ABB RAPID module: GM2698_A.mod

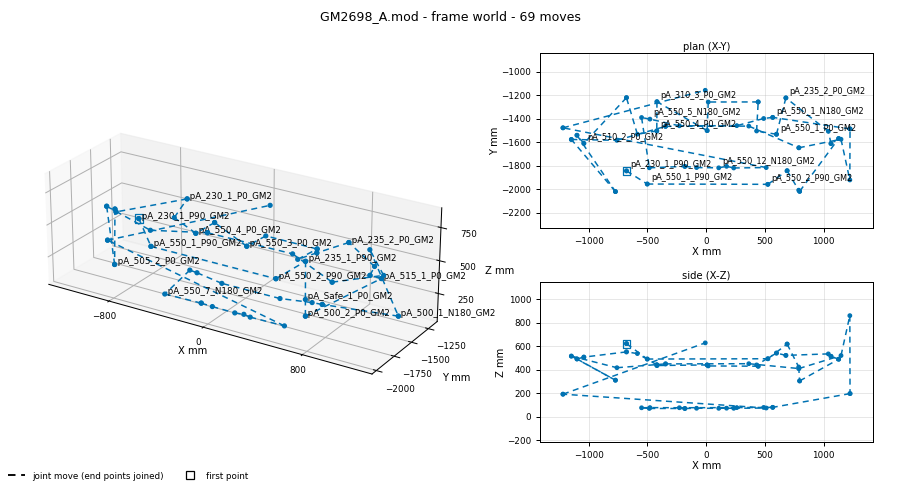
[picture p0: tool path of GM2698_A.mod in frame world, 69 of 75 moves have a stored position in this frame; points joined in program order, loops and branches not executed]
MODULE GM2698_A
!Tool number 7
	TASK PERS wobjdata wobj_A_GM2:=[FALSE,TRUE,"STN2",[[13.9887,-1106.54,385.608],[0.000303697,0.000861464,0.00233511,0.999997]],[[5.18442,-1.41215,-6.83269],[0.999989,-0.00459694,0.000966028,0.00104401]]];

	CONST robtarget pGM2698Tool_A_X1_GM2:=[[548.29,-1104.36,378.90],[0.999992,7.82758E-05,-0.000104085,0.00393794],[-1,0,-1,1],[9E+09,9E+09,9E+09,9E+09,0.0286518,9E+09]];
	CONST robtarget pGM2698Tool_A_X2_GM2:=[[-529.79,-1105.95,378.66],[1,1.60933E-06,-2.29478E-05,2.63453E-05],[-2,-1,0,1],[9E+09,9E+09,9E+09,9E+09,0.0293692,9E+09]];
	CONST robtarget pGM2698Tool_A_Y1_GM2:=[[10.44,-2216.22,373.75],[1,-3.56138E-05,-7.66218E-05,9.50694E-06],[-1,0,-1,1],[9E+09,9E+09,9E+09,9E+09,0.414757,9E+09]];

	!!TRUNNION AT P90
	CONST robtarget pA_230_1_P90_GM2:=[[687.93,736.01,247.05],[8.58268E-05,2.46025E-05,0.000125716,-1],[-2,-1,0,1],[9E+09,9E+09,9E+09,9E+09,89.9785,9E+09]];
	CONST robtarget pA_230_2_P90_GM2:=[[708.26,975.31,-115.95],[0.037863,-0.00102003,-0.000432508,-0.999282],[-2,-1,0,1],[9E+09,9E+09,9E+09,9E+09,44.9633,9E+09]];
	CONST robtarget pA_230_3_P90_GM2:=[[708.26,975.31,-115.95],[0.037863,-0.00102003,-0.000432508,-0.999282],[-2,-1,0,1],[9E+09,9E+09,9E+09,9E+09,44.9633,9E+09]];
	!
	CONST robtarget pA_235_1_P90_GM2:=[[-678.61,736.57,242.76],[0.00931104,0.000190613,-8.92784E-05,0.999957],[-1,0,-1,1],[9E+09,9E+09,9E+09,9E+09,89.9715,9E+09]];
	CONST robtarget pA_235_2_P90_GM2:=[[708.26,975.31,-115.95],[0.037863,-0.00102003,-0.000432508,-0.999282],[-2,-1,0,1],[9E+09,9E+09,9E+09,9E+09,44.9633,9E+09]];
	CONST robtarget pA_235_3_P90_GM2:=[[708.26,975.31,-115.95],[0.037863,-0.00102003,-0.000432508,-0.999282],[-2,-1,0,1],[9E+09,9E+09,9E+09,9E+09,44.9633,9E+09]];
	!
	CONST robtarget pA_310_1_P90_GM2:=[[353.10,729.89,294.43],[0.000108228,5.31787E-05,0.0438261,0.999039],[-2,-1,0,1],[9E+09,9E+09,9E+09,9E+09,89.9716,9E+09]];
	CONST robtarget pA_310_2_P90_GM2:=[[120.58,746.64,293.48],[0.000119282,2.78364E-05,-0.0697897,0.997561],[-2,-1,0,1],[9E+09,9E+09,9E+09,9E+09,89.9659,9E+09]];
	CONST robtarget pA_310_3_P90_GM2:=[[-126.06,745.90,293.24],[8.89304E-05,2.54854E-06,-0.0697908,0.997561],[-1,0,-1,1],[9E+09,9E+09,9E+09,9E+09,89.9658,9E+09]];
	CONST robtarget pA_310_4_P90_GM2:=[[-352.83,729.33,296.03],[0.000103667,2.41673E-05,0.0452051,0.998978],[-1,0,-1,1],[9E+09,9E+09,9E+09,9E+09,89.9674,9E+09]];
	CONST robtarget pA_310_5_P90_GM2:=[[708.26,975.31,-115.95],[0.037863,-0.00102003,-0.000432508,-0.999282],[-2,-1,0,1],[9E+09,9E+09,9E+09,9E+09,44.9633,9E+09]];
	!
	CONST robtarget pA_550_1_P90_GM2:=[[511.36,848.54,116.26],[0.000118797,-6.09284E-05,3.87415E-05,-1],[-2,-1,0,1],[9E+09,9E+09,9E+09,9E+09,89.9792,9E+09]];
	CONST robtarget pA_550_2_P90_GM2:=[[-514.41,852.57,118.58],[0.000364177,0.00017202,0.00027161,-1],[-1,0,-1,1],[9E+09,9E+09,9E+09,9E+09,89.9758,9E+09]];
	CONST robtarget pA_550_3_P90_GM2:=[[335.13,751.81,293.47],[0.000114739,1.47188E-05,-0.069799,0.997561],[-2,-1,0,1],[9E+09,9E+09,9E+09,9E+09,89.9654,9E+09]];
	CONST robtarget pA_550_4_P90_GM2:=[[335.13,751.81,293.47],[0.000114739,1.47188E-05,-0.069799,0.997561],[-2,-1,0,1],[9E+09,9E+09,9E+09,9E+09,89.9654,9E+09]];
	CONST robtarget pA_550_5_P90_GM2:=[[335.13,751.81,293.47],[0.000114739,1.47188E-05,-0.069799,0.997561],[-2,-1,0,1],[9E+09,9E+09,9E+09,9E+09,89.9654,9E+09]];
	CONST robtarget pA_550_6_P90_GM2:=[[335.13,751.81,293.47],[0.000114739,1.47188E-05,-0.069799,0.997561],[-2,-1,0,1],[9E+09,9E+09,9E+09,9E+09,89.9654,9E+09]];
	CONST robtarget pA_550_7_P90_GM2:=[[335.13,751.81,293.47],[0.000114739,1.47188E-05,-0.069799,0.997561],[-2,-1,0,1],[9E+09,9E+09,9E+09,9E+09,89.9654,9E+09]];
	CONST robtarget pA_550_8_P90_GM2:=[[335.13,751.81,293.47],[0.000114739,1.47188E-05,-0.069799,0.997561],[-2,-1,0,1],[9E+09,9E+09,9E+09,9E+09,89.9654,9E+09]];
	CONST robtarget pA_550_9_P90_GM2:=[[335.13,751.81,293.47],[0.000114739,1.47188E-05,-0.069799,0.997561],[-2,-1,0,1],[9E+09,9E+09,9E+09,9E+09,89.9654,9E+09]];
	CONST robtarget pA_550_10_P90_GM2:=[[335.13,751.81,293.47],[0.000114739,1.47188E-05,-0.069799,0.997561],[-2,-1,0,1],[9E+09,9E+09,9E+09,9E+09,89.9654,9E+09]];

	!!TRUNNION AT P0
	CONST robtarget pA_230_1_P0_GM2:=[[687.38,113.52,173.86],[0.00744481,0.444927,0.0139379,-0.895428],[-2,-1,-1,1],[9E+09,9E+09,9E+09,9E+09,-0.0044309,9E+09]];
	CONST robtarget pA_230_2_P0_GM2:=[[714.73,248.80,217.03],[0.0301629,0.281201,0.193711,0.939411],[-2,-2,1,1],[9E+09,9E+09,9E+09,9E+09,14.3078,9E+09]];
	CONST robtarget pA_230_3_P0_GM2:=[[708.26,975.31,-115.95],[0.037863,-0.00102003,-0.000432508,-0.999282],[-2,-1,0,1],[9E+09,9E+09,9E+09,9E+09,44.9633,9E+09]];
	!
	CONST robtarget pA_235_1_P0_GM2:=[[-730.47,258.27,215.19],[0.0469032,0.293033,-0.14088,-0.944503],[-1,1,-2,1],[9E+09,9E+09,9E+09,9E+09,15.4894,9E+09]];
	CONST robtarget pA_235_2_P0_GM2:=[[-668.80,117.45,143.98],[0.00289527,-0.436527,-0.00432652,-0.899677],[-1,0,0,1],[9E+09,9E+09,9E+09,9E+09,-0.011942,9E+09]];
	CONST robtarget pA_235_3_P0_GM2:=[[708.26,975.31,-115.95],[0.037863,-0.00102003,-0.000432508,-0.999282],[-2,-1,0,1],[9E+09,9E+09,9E+09,9E+09,44.9633,9E+09]];
	!
	CONST robtarget pA_310_1_P0_GM2:=[[-433.18,151.92,51.95],[1.60386E-05,5.67962E-05,0.0413145,0.999146],[-1,0,-1,1],[9E+09,9E+09,9E+09,9E+09,-0.0118576,9E+09]];
	CONST robtarget pA_310_2_P0_GM2:=[[-8.33,151.75,54.29],[6.56249E-05,0.000101471,0.0457973,0.998951],[-1,0,-1,1],[9E+09,9E+09,9E+09,9E+09,-0.0110137,9E+09]];
	CONST robtarget pA_310_3_P0_GM2:=[[428.07,148.75,57.96],[2.66549E-05,-6.70695E-06,0.0471647,0.998887],[-2,-1,0,1],[9E+09,9E+09,9E+09,9E+09,-0.00898821,9E+09]];
	CONST robtarget pA_310_4_P0_GM2:=[[708.26,975.31,-115.95],[0.037863,-0.00102003,-0.000432508,-0.999282],[-2,-1,0,1],[9E+09,9E+09,9E+09,9E+09,44.9633,9E+09]];
	CONST robtarget pA_310_5_P0_GM2:=[[708.26,975.31,-115.95],[0.037863,-0.00102003,-0.000432508,-0.999282],[-2,-1,0,1],[9E+09,9E+09,9E+09,9E+09,44.9633,9E+09]];
	!
	CONST robtarget pA_500_1_P0_GM2:=[[-1201.57,789.37,-64.62],[0.00293341,-0.00121104,0.000140597,-0.999995],[-1,0,-1,1],[9E+09,9E+09,9E+09,9E+09,29.7666,9E+09]];
	CONST robtarget pA_500_2_P0_GM2:=[[-784.67,913.62,-69.87],[0.0310443,0.0713657,0.0170151,-0.996822],[-1,0,-1,1],[9E+09,9E+09,9E+09,9E+09,29.7701,9E+09]];
	CONST robtarget pA_500_3_P0_GM2:=[[708.26,975.31,-115.95],[0.037863,-0.00102003,-0.000432508,-0.999282],[-2,-1,0,1],[9E+09,9E+09,9E+09,9E+09,44.9633,9E+09]];
	CONST robtarget pA_500_4_P0_GM2:=[[708.26,975.31,-115.95],[0.037863,-0.00102003,-0.000432508,-0.999282],[-2,-1,0,1],[9E+09,9E+09,9E+09,9E+09,44.9633,9E+09]];
	CONST robtarget pA_500_5_P0_GM2:=[[708.26,975.31,-115.95],[0.037863,-0.00102003,-0.000432508,-0.999282],[-2,-1,0,1],[9E+09,9E+09,9E+09,9E+09,44.9633,9E+09]];
	!
	CONST robtarget pA_505_1_P0_GM2:=[[1202.97,791.70,-68.86],[0.00492061,0.00110187,-4.76185E-05,0.999987],[-2,-1,0,1],[9E+09,9E+09,9E+09,9E+09,29.4165,9E+09]];
	CONST robtarget pA_505_2_P0_GM2:=[[782.38,913.28,-63.33],[0.0152789,0.0774775,-0.00477043,0.996866],[-2,-1,0,1],[9E+09,9E+09,9E+09,9E+09,29.4215,9E+09]];
	CONST robtarget pA_505_3_P0_GM2:=[[708.26,975.31,-115.95],[0.037863,-0.00102003,-0.000432508,-0.999282],[-2,-1,0,1],[9E+09,9E+09,9E+09,9E+09,44.9633,9E+09]];
	CONST robtarget pA_505_4_P0_GM2:=[[708.26,975.31,-115.95],[0.037863,-0.00102003,-0.000432508,-0.999282],[-2,-1,0,1],[9E+09,9E+09,9E+09,9E+09,44.9633,9E+09]];
	CONST robtarget pA_505_5_P0_GM2:=[[708.26,975.31,-115.95],[0.037863,-0.00102003,-0.000432508,-0.999282],[-2,-1,0,1],[9E+09,9E+09,9E+09,9E+09,44.9633,9E+09]];
	!
	CONST robtarget pA_510_1_P0_GM2:=[[1108.89,432.68,115.17],[0.112654,0.176226,0.0162339,0.977748],[-2,-1,1,1],[9E+09,9E+09,9E+09,9E+09,-0.0107183,9E+09]];
	CONST robtarget pA_510_2_P0_GM2:=[[1050.40,501.98,131.19],[0.0176776,-0.325143,0.0102617,0.945444],[-2,-1,-1,1],[9E+09,9E+09,9E+09,9E+09,-0.0104229,9E+09]];
	CONST robtarget pA_510_3_P0_GM2:=[[1153.27,592.76,100.47],[0.0365802,0.172145,-0.0278504,0.983998],[-2,-1,1,1],[9E+09,9E+09,9E+09,9E+09,26.5127,9E+09]];
	CONST robtarget pA_510_4_P0_GM2:=[[1048.95,504.25,129.99],[0.0176891,-0.325131,0.010239,0.945448],[-2,-1,0,1],[9E+09,9E+09,9E+09,9E+09,-0.011562,9E+09]];
	!
	CONST robtarget pA_515_1_P0_GM2:=[[-1117.17,463.93,112.66],[0.108166,0.211616,-0.00270155,-0.971345],[-1,0,-2,1],[9E+09,9E+09,9E+09,9E+09,-0.012828,9E+09]];
	CONST robtarget pA_515_2_P0_GM2:=[[-1052.07,506.56,137.57],[0.000402809,-0.35302,0.000389817,-0.935616],[-1,0,0,1],[9E+09,9E+09,9E+09,9E+09,-0.0197907,9E+09]];
	CONST robtarget pA_515_3_P0_GM2:=[[-1152.24,635.08,93.24],[0.0988859,0.169779,0.00503263,-0.980495],[-1,0,-2,1],[9E+09,9E+09,9E+09,9E+09,36.5012,9E+09]];
	CONST robtarget pA_515_4_P0_GM2:=[[-1045.41,506.20,133.06],[0.000367603,-0.353062,0.000351063,-0.9356],[-1,0,0,1],[9E+09,9E+09,9E+09,9E+09,-0.0197905,9E+09]];
	!
	CONST robtarget pA_520_1_P0_GM2:=[[708.26,975.31,-115.95],[0.037863,-0.00102003,-0.000432508,-0.999282],[-2,-1,0,1],[9E+09,9E+09,9E+09,9E+09,44.9633,9E+09]];
	CONST robtarget pA_520_2_P0_GM2:=[[708.26,975.31,-115.95],[0.037863,-0.00102003,-0.000432508,-0.999282],[-2,-1,0,1],[9E+09,9E+09,9E+09,9E+09,44.9633,9E+09]];
	CONST robtarget pA_520_3_P0_GM2:=[[708.26,975.31,-115.95],[0.037863,-0.00102003,-0.000432508,-0.999282],[-2,-1,0,1],[9E+09,9E+09,9E+09,9E+09,44.9633,9E+09]];
	CONST robtarget pA_520_4_P0_GM2:=[[708.26,975.31,-115.95],[0.037863,-0.00102003,-0.000432508,-0.999282],[-2,-1,0,1],[9E+09,9E+09,9E+09,9E+09,44.9633,9E+09]];
	CONST robtarget pA_520_5_P0_GM2:=[[708.26,975.31,-115.95],[0.037863,-0.00102003,-0.000432508,-0.999282],[-2,-1,0,1],[9E+09,9E+09,9E+09,9E+09,44.9633,9E+09]];
	!
	CONST robtarget pA_550_1_P0_GM2:=[[-588.27,426.70,164.89],[0.0152053,0.548166,0.0110567,0.836158],[-2,0,0,1],[9E+09,9E+09,9E+09,9E+09,-0.0169634,9E+09]];
	CONST robtarget pA_550_2_P0_GM2:=[[-419.34,398.83,64.09],[1.55675E-05,-3.99913E-05,1.7675E-05,1],[-1,0,-1,1],[9E+09,9E+09,9E+09,9E+09,-0.0173011,9E+09]];
	CONST robtarget pA_550_3_P0_GM2:=[[1.46,395.01,63.93],[1.08108E-05,-9.40457E-06,-2.05058E-05,-1],[-1,0,-1,1],[9E+09,9E+09,9E+09,9E+09,-0.022618,9E+09]];
	CONST robtarget pA_550_4_P0_GM2:=[[429.81,397.20,65.70],[8.27019E-06,8.95741E-05,-5.33681E-05,1],[-2,-1,0,1],[9E+09,9E+09,9E+09,9E+09,-0.0133345,9E+09]];
	CONST robtarget pA_550_5_P0_GM2:=[[594.89,424.65,160.92],[0.028073,0.537019,-0.0220339,-0.842814],[-1,-1,-1,1],[9E+09,9E+09,9E+09,9E+09,-0.0155708,9E+09]];
	CONST robtarget pA_550_6_P0_GM2:=[[708.26,975.31,-115.95],[0.037863,-0.00102003,-0.000432508,-0.999282],[-2,-1,0,1],[9E+09,9E+09,9E+09,9E+09,44.9633,9E+09]];
	CONST robtarget pA_550_7_P0_GM2:=[[708.26,975.31,-115.95],[0.037863,-0.00102003,-0.000432508,-0.999282],[-2,-1,0,1],[9E+09,9E+09,9E+09,9E+09,44.9633,9E+09]];
	CONST robtarget pA_550_8_P0_GM2:=[[708.26,975.31,-115.95],[0.037863,-0.00102003,-0.000432508,-0.999282],[-2,-1,0,1],[9E+09,9E+09,9E+09,9E+09,44.9633,9E+09]];
	CONST robtarget pA_550_9_P0_GM2:=[[708.26,975.31,-115.95],[0.037863,-0.00102003,-0.000432508,-0.999282],[-2,-1,0,1],[9E+09,9E+09,9E+09,9E+09,44.9633,9E+09]];
	CONST robtarget pA_550_10_P0_GM2:=[[708.26,975.31,-115.95],[0.037863,-0.00102003,-0.000432508,-0.999282],[-2,-1,0,1],[9E+09,9E+09,9E+09,9E+09,44.9633,9E+09]];
	!
	!!TRUNNION AT N60
	CONST robtarget pA_500_1_N60_GM2:=[[-778.58,542.42,33.75],[0.00280107,0.0438531,0.00715282,-0.999009],[-1,0,-1,1],[9E+09,9E+09,9E+09,9E+09,-60.5132,9E+09]];
	CONST robtarget pA_500_2_N60_GM2:=[[-1217.46,473.19,8.92],[0.00374905,-0.104264,0.00695893,-0.994518],[-1,0,-1,1],[9E+09,9E+09,9E+09,9E+09,-60.5084,9E+09]];
	CONST robtarget pA_500_3_N60_GM2:=[[-1137.33,470.02,143.84],[0.00403999,-0.000135764,2.34192E-05,-0.999992],[-1,0,-1,1],[9E+09,9E+09,9E+09,9E+09,-60.5103,9E+09]];
	CONST robtarget pA_500_4_N60_GM2:=[[708.26,975.31,-115.95],[0.037863,-0.00102003,-0.000432508,-0.999282],[-2,-1,0,1],[9E+09,9E+09,9E+09,9E+09,44.9633,9E+09]];
	CONST robtarget pA_500_5_N60_GM2:=[[708.26,975.31,-115.95],[0.037863,-0.00102003,-0.000432508,-0.999282],[-2,-1,0,1],[9E+09,9E+09,9E+09,9E+09,44.9633,9E+09]];
	!
	CONST robtarget pA_505_1_N60_GM2:=[[1156.75,468.38,139.62],[0.00522979,-1.17706E-05,-7.50595E-05,-0.999987],[-2,-1,0,1],[9E+09,9E+09,9E+09,9E+09,-60.5089,9E+09]];
	CONST robtarget pA_505_2_N60_GM2:=[[1216.37,472.20,8.95],[0.00194678,0.139228,0.00768064,-0.990228],[-2,-1,0,1],[9E+09,9E+09,9E+09,9E+09,-60.506,9E+09]];
	CONST robtarget pA_505_3_N60_GM2:=[[769.08,476.65,40.85],[0.0019964,-0.0777815,-8.25469E-05,-0.996969],[-2,-1,0,1],[9E+09,9E+09,9E+09,9E+09,-60.5041,9E+09]];
	CONST robtarget pA_505_4_N60_GM2:=[[708.26,975.31,-115.95],[0.037863,-0.00102003,-0.000432508,-0.999282],[-2,-1,0,1],[9E+09,9E+09,9E+09,9E+09,44.9633,9E+09]];
	CONST robtarget pA_505_5_N60_GM2:=[[708.26,975.31,-115.95],[0.037863,-0.00102003,-0.000432508,-0.999282],[-2,-1,0,1],[9E+09,9E+09,9E+09,9E+09,44.9633,9E+09]];
	!
	CONST robtarget pA_520_1_N60_GM2:=[[355.07,358.37,72.76],[0.00521062,-0.000565034,0.105165,-0.994441],[-2,-1,0,1],[9E+09,9E+09,9E+09,9E+09,-60.5116,9E+09]];
	CONST robtarget pA_520_2_N60_GM2:=[[-123.90,988.17,-108.46],[0.000713776,4.54184E-05,8.43669E-05,-0.999999],[-1,0,-1,1],[9E+09,9E+09,9E+09,9E+09,60.0162,9E+09]];
	CONST robtarget pA_520_3_N60_GM2:=[[123.84,989.35,-108.45],[0.000730733,6.40844E-05,7.66397E-05,-0.999999],[-2,-1,0,1],[9E+09,9E+09,9E+09,9E+09,60.0163,9E+09]];
	CONST robtarget pA_520_4_N60_GM2:=[[-353.01,357.21,74.17],[0.00521171,-0.000602148,0.105152,-0.994442],[-1,0,-1,1],[9E+09,9E+09,9E+09,9E+09,-60.5086,9E+09]];
	!
	!!TRUNNION AT N180
	!
	CONST robtarget pA_310_1_N180_GM2:=[[-427.01,928.00,-352.17],[4.23949E-05,1.23545E-06,-0.117062,-0.993125],[-1,0,-1,1],[9E+09,9E+09,9E+09,9E+09,-171.335,9E+09]];
	CONST robtarget pA_310_2_N180_GM2:=[[-341.86,937.73,-374.62],[1.08478E-05,-1.53197E-05,6.13881E-05,-1],[-1,0,-1,1],[9E+09,9E+09,9E+09,9E+09,-171.333,9E+09]];
	CONST robtarget pA_310_3_N180_GM2:=[[-161.23,931.93,-349.80],[8.00821E-06,-4.37144E-05,-0.117485,-0.993075],[-1,0,-1,1],[9E+09,9E+09,9E+09,9E+09,-171.335,9E+09]];
	CONST robtarget pA_310_4_N180_GM2:=[[9.06,936.16,-374.68],[2.71618E-05,-1.9313E-05,-0.0604457,-0.998172],[-2,-1,0,1],[9E+09,9E+09,9E+09,9E+09,-171.334,9E+09]];
	CONST robtarget pA_310_5_N180_GM2:=[[157.83,928.08,-351.40],[4.23165E-05,-2.36973E-05,-0.117106,-0.99312],[-2,-1,0,1],[9E+09,9E+09,9E+09,9E+09,-171.335,9E+09]];
	CONST robtarget pA_310_6_N180_GM2:=[[431.92,925.50,-350.73],[4.91988E-05,-7.21662E-05,-0.117557,-0.993066],[-2,-1,0,1],[9E+09,9E+09,9E+09,9E+09,-171.335,9E+09]];
	CONST robtarget pA_310_7_N180_GM2:=[[492.88,939.60,-374.19],[4.56863E-05,-1.05492E-05,6.13342E-05,-1],[-2,-1,0,1],[9E+09,9E+09,9E+09,9E+09,-171.333,9E+09]];
	CONST robtarget pA_310_8_N180_GM2:=[[708.26,975.31,-115.95],[0.037863,-0.00102003,-0.000432508,-0.999282],[-2,-1,0,1],[9E+09,9E+09,9E+09,9E+09,44.9633,9E+09]];
	CONST robtarget pA_310_9_N180_GM2:=[[708.26,975.31,-115.95],[0.037863,-0.00102003,-0.000432508,-0.999282],[-2,-1,0,1],[9E+09,9E+09,9E+09,9E+09,44.9633,9E+09]];
	CONST robtarget pA_310_10_N180_GM2:=[[708.26,975.31,-115.95],[0.037863,-0.00102003,-0.000432508,-0.999282],[-2,-1,0,1],[9E+09,9E+09,9E+09,9E+09,44.9633,9E+09]];
	CONST robtarget pA_310_11_N180_GM2:=[[708.26,975.31,-115.95],[0.037863,-0.00102003,-0.000432508,-0.999282],[-2,-1,0,1],[9E+09,9E+09,9E+09,9E+09,44.9633,9E+09]];
	CONST robtarget pA_310_12_N180_GM2:=[[708.26,975.31,-115.95],[0.037863,-0.00102003,-0.000432508,-0.999282],[-2,-1,0,1],[9E+09,9E+09,9E+09,9E+09,44.9633,9E+09]];
	CONST robtarget pA_310_13_N180_GM2:=[[708.26,975.31,-115.95],[0.037863,-0.00102003,-0.000432508,-0.999282],[-2,-1,0,1],[9E+09,9E+09,9E+09,9E+09,44.9633,9E+09]];
	CONST robtarget pA_310_14_N180_GM2:=[[708.26,975.31,-115.95],[0.037863,-0.00102003,-0.000432508,-0.999282],[-2,-1,0,1],[9E+09,9E+09,9E+09,9E+09,44.9633,9E+09]];
	CONST robtarget pA_310_15_N180_GM2:=[[708.26,975.31,-115.95],[0.037863,-0.00102003,-0.000432508,-0.999282],[-2,-1,0,1],[9E+09,9E+09,9E+09,9E+09,44.9633,9E+09]];

	!
	CONST robtarget pA_500_1_N180_GM2:=[[-1214.15,383.59,-180.12],[0.706069,-6.54173E-05,-1.71735E-05,-0.708144],[-1,-1,0,1],[9E+09,9E+09,9E+09,9E+09,-149.959,9E+09]];
	CONST robtarget pA_500_2_N180_GM2:=[[-1204.66,381.86,-186.15],[0.32853,-6.5977E-06,4.28364E-05,-0.944493],[-1,0,-1,1],[9E+09,9E+09,9E+09,9E+09,-149.952,9E+09]];
	CONST robtarget pA_500_3_N180_GM2:=[[-1137.07,519.96,141.43],[0.00405737,-1.80252E-05,5.82048E-05,-0.999991],[-1,0,-1,1],[9E+09,9E+09,9E+09,9E+09,-60.5062,9E+09]];
	CONST robtarget pA_500_4_N180_GM2:=[[708.26,975.31,-115.95],[0.037863,-0.00102003,-0.000432508,-0.999282],[-2,-1,0,1],[9E+09,9E+09,9E+09,9E+09,44.9633,9E+09]];
	CONST robtarget pA_500_5_N180_GM2:=[[708.26,975.31,-115.95],[0.037863,-0.00102003,-0.000432508,-0.999282],[-2,-1,0,1],[9E+09,9E+09,9E+09,9E+09,44.9633,9E+09]];
	!
	CONST robtarget pA_505_1_N180_GM2:=[[1227.95,370.76,-184.70],[0.703813,2.0347E-05,-0.000363019,0.710385],[-2,0,-1,1],[9E+09,9E+09,9E+09,9E+09,-149.954,9E+09]];
	CONST robtarget pA_505_2_N180_GM2:=[[1191.41,389.44,-184.88],[0.320474,-4.84084E-05,-0.000382623,0.947257],[-2,-1,0,1],[9E+09,9E+09,9E+09,9E+09,-149.948,9E+09]];
	CONST robtarget pA_505_3_N180_GM2:=[[775.04,447.88,42.59],[0.00201212,-0.0777562,-8.91676E-05,-0.99697],[-2,-1,0,1],[9E+09,9E+09,9E+09,9E+09,-60.5045,9E+09]];
	CONST robtarget pA_505_4_N180_GM2:=[[708.26,975.31,-115.95],[0.037863,-0.00102003,-0.000432508,-0.999282],[-2,-1,0,1],[9E+09,9E+09,9E+09,9E+09,44.9633,9E+09]];
	CONST robtarget pA_505_5_N180_GM2:=[[708.26,975.31,-115.95],[0.037863,-0.00102003,-0.000432508,-0.999282],[-2,-1,0,1],[9E+09,9E+09,9E+09,9E+09,44.9633,9E+09]];
	!
	CONST robtarget pA_550_1_N180_GM2:=[[-556.66,284.95,-297.43],[0.0146441,-0.000738703,-0.0640003,-0.997842],[-1,0,-1,1],[9E+09,9E+09,9E+09,9E+09,-179.982,9E+09]];
	CONST robtarget pA_550_2_N180_GM2:=[[-479.54,294.52,-298.21],[0.0147177,0.000968414,-0.0648092,-0.997788],[-1,0,-1,1],[9E+09,9E+09,9E+09,9E+09,-179.974,9E+09]];
	CONST robtarget pA_550_3_N180_GM2:=[[-250.78,354.86,-299.12],[0.00839662,0.00062424,-0.0673719,-0.997693],[-1,0,-1,1],[9E+09,9E+09,9E+09,9E+09,-179.978,9E+09]];
	CONST robtarget pA_550_4_N180_GM2:=[[237.67,355.52,-300.25],[0.006963,0.000448698,-0.0699319,-0.997528],[-2,-1,0,1],[9E+09,9E+09,9E+09,9E+09,-179.971,9E+09]];
	CONST robtarget pA_550_5_N180_GM2:=[[488.03,298.32,-299.34],[0.0147834,0.00108507,-0.0688852,-0.997515],[-2,-1,0,1],[9E+09,9E+09,9E+09,9E+09,-179.978,9E+09]];
	CONST robtarget pA_550_6_N180_GM2:=[[559.15,284.61,-300.90],[0.0147563,0.000914124,-0.0621348,-0.997959],[-2,-1,0,1],[9E+09,9E+09,9E+09,9E+09,-179.972,9E+09]];
	CONST robtarget pA_550_7_N180_GM2:=[[493.82,712.51,-304.58],[0.00369609,1.44225E-05,-0.000177454,0.999993],[-2,-1,0,1],[9E+09,9E+09,9E+09,9E+09,-179.978,9E+09]];
	CONST robtarget pA_550_8_N180_GM2:=[[191.37,701.01,-305.16],[0.000471327,-4.0688E-05,2.47394E-05,-1],[-2,-1,0,1],[9E+09,9E+09,9E+09,9E+09,-179.98,9E+09]];
	CONST robtarget pA_550_9_N180_GM2:=[[162.52,714.71,-304.99],[0.00044817,-2.64542E-05,3.82305E-05,-1],[-2,-1,0,1],[9E+09,9E+09,9E+09,9E+09,-179.977,9E+09]];
	CONST robtarget pA_550_10_N180_GM2:=[[92.00,710.92,-303.09],[0.000492036,-8.80391E-06,3.65271E-05,-1],[-2,-1,0,1],[9E+09,9E+09,9E+09,9E+09,-179.979,9E+09]];
	CONST robtarget pA_550_11_N180_GM2:=[[-2.18,734.80,-301.09],[0.000503616,-3.449E-05,2.8216E-05,-0.999999],[-2,0,-1,1],[9E+09,9E+09,9E+09,9E+09,-179.976,9E+09]];
	CONST robtarget pA_550_12_N180_GM2:=[[-96.61,713.50,-303.62],[0.000531659,-1.04945E-05,2.9268E-05,-1],[-1,0,-1,1],[9E+09,9E+09,9E+09,9E+09,-179.979,9E+09]];
	CONST robtarget pA_550_13_N180_GM2:=[[-163.24,700.92,-302.64],[0.000557157,-1.5553E-06,6.84997E-06,-1],[-1,0,-1,1],[9E+09,9E+09,9E+09,9E+09,-179.984,9E+09]];
	CONST robtarget pA_550_14_N180_GM2:=[[-224.30,714.89,-303.47],[0.000565679,-1.66874E-05,-1.44057E-05,-1],[-1,0,-1,1],[9E+09,9E+09,9E+09,9E+09,-179.982,9E+09]];
	CONST robtarget pA_550_15_N180_GM2:=[[-500.65,711.97,-301.26],[0.00055817,-3.54601E-05,1.56352E-05,-1],[-1,0,-1,1],[9E+09,9E+09,9E+09,9E+09,-179.988,9E+09]];
	CONST robtarget pA_550_16_N180_GM2:=[[335.13,751.81,293.47],[0.000114739,1.47188E-05,-0.069799,0.997561],[-2,-1,0,1],[9E+09,9E+09,9E+09,9E+09,89.9654,9E+09]];
	CONST robtarget pA_550_17_N180_GM2:=[[335.13,751.81,293.47],[0.000114739,1.47188E-05,-0.069799,0.997561],[-2,-1,0,1],[9E+09,9E+09,9E+09,9E+09,89.9654,9E+09]];
	CONST robtarget pA_550_18_N180_GM2:=[[335.13,751.81,293.47],[0.000114739,1.47188E-05,-0.069799,0.997561],[-2,-1,0,1],[9E+09,9E+09,9E+09,9E+09,89.9654,9E+09]];
	CONST robtarget pA_550_19_N180_GM2:=[[351.91,756.93,-300.99],[0.0147766,-2.34032E-05,6.93973E-05,-0.99989],[-2,-1,0,1],[9E+09,9E+09,9E+09,9E+09,-179.977,9E+09]];
	CONST robtarget pA_550_20_N180_GM2:=[[122.27,635.67,-305.15],[0.000474668,-1.23285E-05,1.97455E-05,-1],[-2,-1,0,1],[9E+09,9E+09,9E+09,9E+09,-179.978,9E+09]];
	CONST robtarget pA_550_21_N180_GM2:=[[-128.60,758.45,-301.12],[0.000539466,-5.17921E-06,1.67757E-05,-0.999999],[-1,0,-1,1],[9E+09,9E+09,9E+09,9E+09,-179.978,9E+09]];
	CONST robtarget pA_550_22_N180_GM2:=[[-356.72,760.25,-301.19],[0.000574946,-3.24014E-06,3.82912E-06,-0.999999],[-1,0,-1,1],[9E+09,9E+09,9E+09,9E+09,-179.98,9E+09]];


    TASK PERS loaddata LoadGM2698A:=[900,[-186.8,43.5,0],[1,0,0,0],0,0,111.6];


	CONST robtarget pA_Safe_1_P0_GM2:=[[-776.79,903.09,48.71],[0.0270915,0.0665119,0.0157283,-0.997294],[-1,0,-1,1],[9E+09,9E+09,9E+09,9E+09,31.3258,9E+09]];
	CONST robtarget pA_Safe_2_P0_GM2:=[[-1173.26,505.55,308.17],[0.299253,-0.00605452,0.0185665,-0.953974],[-1,0,-1,1],[9E+09,9E+09,9E+09,9E+09,-0.0127436,9E+09]];
	CONST robtarget pA_Safe_3_P0_GM2:=[[1206.65,483.09,309.68],[0.320571,-0.00610917,-0.0189757,0.947014],[-2,0,-1,1],[9E+09,9E+09,9E+09,9E+09,-0.012828,9E+09]];
	CONST robtarget pA_Safe_4_P0_GM2:=[[-867.31,489.74,258.29],[0.0101084,2.8178E-05,-5.44035E-05,0.999949],[-1,0,-1,1],[9E+09,9E+09,9E+09,9E+09,-0.012828,9E+09]];
	CONST robtarget pA_Safe_5_P0_GM2:=[[-867.31,489.74,258.29],[0.0101084,2.8178E-05,-5.44035E-05,0.999949],[-1,0,-1,1],[9E+09,9E+09,9E+09,9E+09,-0.012828,9E+09]];
	CONST robtarget pA_Safe_6_P0_GM2:=[[-867.31,489.74,258.29],[0.0101084,2.8178E-05,-5.44035E-05,0.999949],[-1,0,-1,1],[9E+09,9E+09,9E+09,9E+09,-0.012828,9E+09]];
	CONST robtarget pA_Safe_7_P0_GM2:=[[-867.31,489.74,258.29],[0.0101084,2.8178E-05,-5.44035E-05,0.999949],[-1,0,-1,1],[9E+09,9E+09,9E+09,9E+09,-0.012828,9E+09]];

	CONST robtarget pA_Safe_1_N180_GM2:=[[-1211.92,814.58,484.94],[0.113943,-0.0335182,0.225338,-0.967015],[-1,0,-1,1],[9E+09,9E+09,9E+09,9E+09,-62.6189,9E+09]];
	CONST robtarget pA_Safe_2_N180_GM2:=[[16.89,51.24,250.08],[0.00136107,-3.49227E-05,0.000388549,-0.999999],[-2,-1,0,1],[9E+09,9E+09,9E+09,9E+09,-149.948,9E+09]];
	CONST robtarget pA_Safe_3_N180_GM2:=[[16.88,51.24,250.08],[0.00136295,-3.96608E-05,0.000388216,-0.999999],[-2,-1,0,1],[9E+09,9E+09,9E+09,9E+09,33.5415,9E+09]];

	CONST robtarget pA_445_safe01_N180_GM2:=[[-1030.14,449.69,-57.42],[0.139634,-0.000906499,-0.000277604,-0.990202],[-1,0,-1,1],[9E+09,9E+09,9E+09,9E+09,-179.929,9E+09]];
	CONST robtarget pA_Safe_N90_2_GM2:=[[758.90,24.14,-68.10],[0.000305872,0.00120705,0.173796,0.98478],[-2,-1,0,1],[9E+09,9E+09,9E+09,9E+09,-58.1628,9E+09]];
	CONST robtarget pA_Safe_N90_3_GM2:=[[-894.81,518.59,346.96],[0.00406077,-2.99968E-05,5.05023E-05,-0.999991],[-1,0,-1,1],[9E+09,9E+09,9E+09,9E+09,-60.5068,9E+09]];
	CONST robtarget pA_Safe_1_P0_GM12:=[[-543.62,820.17,65.05],[5.02587E-05,0.000307266,5.46968E-06,1],[-1,0,-1,1],[9E+09,9E+09,9E+09,9E+09,-0.0227023,9E+09]];
	CONST robtarget pA_550_3_P0_GM12:=[[545.82,817.89,57.34],[2.78437E-05,0.000245156,0.000100892,1],[-2,-1,0,1],[9E+09,9E+09,9E+09,9E+09,-0.0315638,9E+09]];
	CONST robtarget pA_500_1_N180_GM12:=[[-1129.50,619.60,-361.57],[0.0233784,0.216958,0.0182336,0.97573],[-1,0,-1,1],[9E+09,9E+09,9E+09,9E+09,-178.615,9E+09]];
	CONST robtarget pA_515_1_P0_GM12:=[[-1117.17,463.93,112.66],[0.108168,0.211621,-0.00269871,-0.971344],[-1,0,-2,1],[9E+09,9E+09,9E+09,9E+09,-0.0123203,9E+09]];
	CONST robtarget pA_550_3_P0_GM22:=[[116.06,395.94,63.70],[3.88215E-05,-1.77326E-05,1.06229E-05,-1],[-2,-1,0,1],[9E+09,9E+09,9E+09,9E+09,-0.0232087,9E+09]];
	CONST robtarget pA_Safe_1_P0_GM22:=[[-116.20,396.03,64.22],[3.20058E-05,-2.53767E-05,1.70392E-05,-1],[-1,0,-1,1],[9E+09,9E+09,9E+09,9E+09,-0.0232087,9E+09]];
	CONST robtarget pA_515_2_P0_GM12:=[[-1029.51,402.17,157.71],[0.000353747,-0.353072,0.000348763,-0.935597],[-1,0,0,1],[9E+09,9E+09,9E+09,9E+09,-0.0192,9E+09]];




	PROC rGM2698_A_Welding()
			SetGO TaskActive, 1;
			rSpeed_Override;
			ClkReset clock_A_Weld_cycle;
			ClkStart clock_A_Weld_cycle;
			PulseDO\PLength:=2.0, WeldStarted;
			!
			PulseDO\PLength:=2.0, OpenCellAInnerDoor;

			ActUnit STN2;
			!DeactUnit STN1;
			MechUnitLoad Stn2, 1, LoadGM2698A;
			WaitDI CellAInnerDoorOpened ,1;
			!

		IF RobotProduction = 1 THEN
			vProduction := [7500,7500,7500,180];
			vHome := [3500, 3500, 3500, 90];
	  	ELSE
			vProduction := [200,100,100,20];
			vHome := [100, 100, 100, 10];
	  	ENDIF
			!
			WaitDI TAClampsSafePFO,1;
			rMoveToCell_A;
			Set PFOAirJet;
			!
			MoveAbsJ pA_Load\NoEOffs, vProduction, z200, t3D_PFO\WObj:=wobj0;
			PulseDO WeldStarted;
			Set LaserRequest;
			IF TAClampsSafePFO = 0 Stop;
			!
			AccSet 100,100;

			!**************************************************
			!Positioner at +90 degree
			!**************************************************
			MoveJ pA_230_1_P90_GM2,vProduction,fine,t3D_PFO\WObj:=wobj_A_GM2;
			IF AS350_1PP = 1 THEN !!!TA230XPP = 1 Then
			!K2 SP
			SetGO PFOProgReq, 312;
			SetGO LaserProgReq, 140;
			MoveJ pA_230_1_P90_GM2,vProduction,fine,t3D_PFO\WObj:=wobj_A_GM2;
			rPFO_Welding;
			!
			ENDIF
			!
			MoveJ pA_550_1_P90_GM2,vProduction,fine,t3D_PFO\WObj:=wobj_A_GM2;
			IF AW550PP = 1 THEN  !!! TA550PP = 1 Then
			!
			!K2 WD
			SetGO PFOProgReq, 112;
			SetGO LaserProgReq, 140;
			MoveJ pA_550_1_P90_GM2,vProduction,fine,t3D_PFO\WObj:=wobj_A_GM2;
			rPFO_Welding;
			!
			ENDIF

			MoveJ pA_550_2_P90_GM2,vProduction,fine,t3D_PFO\WObj:=wobj_A_GM2;
			IF AW550PP = 1 THEN  !!! TA550PP = 1 Then
			!
			!M2 WD
			SetGO PFOProgReq, 118;
			SetGO LaserProgReq, 140;
			MoveJ pA_550_2_P90_GM2,vProduction,fine,t3D_PFO\WObj:=wobj_A_GM2;
			rPFO_Welding;
			!
			ENDIF


			MoveJ pA_235_1_P90_GM2,vProduction,fine,t3D_PFO\WObj:=wobj_A_GM2;
			IF AS350_2PP = 1 THEN !!!  TA235XPP = 1 Then
			!M2 SP
			SetGO PFOProgReq, 318;
			SetGO LaserProgReq, 140;
			MoveJ pA_235_1_P90_GM2,vProduction,fine,t3D_PFO\WObj:=wobj_A_GM2;
			rPFO_Welding;
			!
			ENDIF
			!**************************************************
			!Trunnion at +0 degree
			!*************************************************

			MoveJ pA_Safe_1_P0_GM2, vProduction, z200, t3D_PFO\WObj:=wobj_A_GM2;

			MoveJ pA_500_2_P0_GM2,vProduction,fine,t3D_PFO\WObj:=wobj_A_GM2;
			IF AW500PP = 1 THEN !!! TA500PP = 1 Then

			!H5 WD
			SetGO PFOProgReq, 99;
			SetGO LaserProgReq, 140;
			MoveJ pA_500_2_P0_GM2,vProduction,fine,t3D_PFO\WObj:=wobj_A_GM2;
			rPFO_Welding;

			ENDIF
			!
			MoveJ pA_515_1_P0_GM2,vProduction,fine,t3D_PFO\WObj:=wobj_A_GM2;
			IF AW510_2PP = 1 THEN !!!  TA515 = 1 Then
			!
			!G1 G2-1 G2-2 WD
			SetGO LaserProgReq, 147;
			MoveJ pA_515_1_P0_GM2,vProduction,fine,t3D_PFO\WObj:=wobj_A_GM2;
			rPFO_Welding;
			!WaitTime 1.0;

			ENDIF


		MoveJ pA_515_2_P0_GM2, vProduction, fine, t3D_PFO\WObj:=wobj_A_GM2;
			IF AW510_2PP = 1 THEN !!!  TA515 = 1 Then

			!G3 WD
			SetGO PFOProgReq, 92;
			SetGO LaserProgReq, 140;
			MoveJ pA_515_2_P0_GM2, vProduction, fine, t3D_PFO\WObj:=wobj_A_GM2;
			rPFO_Welding;

			MoveJ pA_515_2_P0_GM12, vPRODUCTION, z200, t3D_PFO\WObj:=wobj_A_GM2;
			!
			ENDIF

			MoveJ pA_235_2_P0_GM2,vProduction,fine,t3D_PFO\WObj:=wobj_A_GM2;
			IF AS350_2PP = 1 THEN !!!  TA235XPP = 1 Then

			!F6 F7 F8 F9 F10
			SetGO LaserProgReq, 149;
			MoveJ pA_235_2_P0_GM2,vProduction,fine,t3D_PFO\WObj:=wobj_A_GM2;
			rPFO_Welding;
			!
			ENDIF

			MoveJ pA_550_1_P0_GM2,vProduction,fine,t3D_PFO\WObj:=wobj_A_GM2;
			IF AW550PP = 1 THEN  !!! TA550PP = 1 Then
			!
			!M3 M4 WD
			SetGO LaserProgReq, 161;
			MoveJ pA_550_1_P0_GM2,vProduction,fine,t3D_PFO\WObj:=wobj_A_GM2;
			rPFO_Welding;
			!
			!M1
			SetGO PFOProgReq, 117;
			SetGO LaserProgReq, 140;
			MoveJ pA_550_2_P0_GM2,vProduction,fine,t3D_PFO\WObj:=wobj_A_GM2;
			rPFO_Welding;
			!
			ENDIF

			MoveJ pA_310_1_P0_GM2,vProduction,fine,t3D_PFO\WObj:=wobj_A_GM2;

			IF AS310PP = 1 THEN !!! TA310XPP = 1 Then
			!K1 SP
			SetGO PFOProgReq, 311;
			SetGO LaserProgReq, 140;
			MoveJ pA_310_1_P0_GM2,vProduction,fine,t3D_PFO\WObj:=wobj_A_GM2;
			rPFO_Welding;
			!
			!J1 J2 SP
			SetGO PFOProgReq, 302;
			SetGO LaserProgReq, 140;
			MoveJ pA_310_2_P0_GM2,vProduction,fine,t3D_PFO\WObj:=wobj_A_GM2;
			rPFO_Welding;

			ENDIF

			MoveJ pA_550_3_P0_GM2,vProduction,fine,t3D_PFO\WObj:=wobj_A_GM2;
			IF AW550PP = 1 THEN  !!! TA550PP = 1 Then

			!J1 J2 WD
			SetGO LaserProgReq, 163;
			MoveJ pA_550_3_P0_GM2,vProduction,fine,t3D_PFO\WObj:=wobj_A_GM2;
			rPFO_Welding;

			ENDIF

			MoveJ pA_310_3_P0_GM2,vProduction,fine,t3D_PFO\WObj:=wobj_A_GM2;
			IF AS310PP = 1 THEN !!! TA310XPP = 1 Then
			!
			SetGO PFOProgReq, 317;
			SetGO LaserProgReq, 140;
			MoveJ pA_310_3_P0_GM2,vProduction,fine,t3D_PFO\WObj:=wobj_A_GM2;
			rPFO_Welding;
			!
			ENDIF

			MoveJ pA_550_4_P0_GM2,vProduction,fine,t3D_PFO\WObj:=wobj_A_GM2;
			IF AW550PP = 1 THEN  !!! TA550PP = 1 Then
			!
			!K1 WD
			SetGO PFOProgReq, 111;
			SetGO LaserProgReq, 140;
			MoveJ pA_550_4_P0_GM2,vProduction,fine,t3D_PFO\WObj:=wobj_A_GM2;
			rPFO_Welding;
			!
			!K3 K4 WD
			SetGO LaserProgReq, 162;
			MoveJ pA_550_5_P0_GM2,vProduction,fine,t3D_PFO\WObj:=wobj_A_GM2;
			rPFO_Welding;
			!
			ENDIF

			MoveJ pA_230_1_P0_GM2,vProduction,fine,t3D_PFO\WObj:=wobj_A_GM2;
			IF AS350_1PP = 1 THEN !!!TA230XPP = 1 Then
			!
			!C6 C7 C8 C9 C10 SP
			SetGO LaserProgReq, 150;
			MoveJ pA_230_1_P0_GM2,vProduction,fine,t3D_PFO\WObj:=wobj_A_GM2;
			rPFO_Welding;

			ENDIF

			MoveJ pA_510_2_P0_GM2, vProduction, fine, t3D_PFO\WObj:=wobj_A_GM2;
			IF AW510_1PP = 1 THEN !!!

			!D3 WD
			SetGO PFOProgReq, 70;
			SetGO LaserProgReq, 140;
			MoveJ pA_510_2_P0_GM2, vProduction, fine, t3D_PFO\WObj:=wobj_A_GM2;
			rPFO_Welding;
			!
			ENDIF

			MoveJ pA_510_1_P0_GM2,vProduction,fine,t3D_PFO\WObj:=wobj_A_GM2;
			IF AW510_1PP = 1 THEN !!!

			!D1 D2-1 D2-2 WD
			SetGO LaserProgReq, 151;
			MoveJ pA_510_1_P0_GM2,vProduction,fine,t3D_PFO\WObj:=wobj_A_GM2;
			rPFO_Welding;

			ENDIF

			MoveJ pA_505_2_P0_GM2,vProduction,fine,t3D_PFO\WObj:=wobj_A_GM2;
			IF AW505PP = 1 THEN  !!! TA505PP = 1 Then

			!E5 WD
			SetGO PFOProgReq, 77;
			SetGO LaserProgReq, 140;
			MoveJ pA_505_2_P0_GM2,vProduction,fine,t3D_PFO\WObj:=wobj_A_GM2;
			rPFO_Welding;

			ENDIF

			!**************************************************
			!Trunnion at -60 degree
			!**************************************************

		MoveJ pA_505_1_N60_GM2,vProduction,fine,t3D_PFO\WObj:=wobj_A_GM2;
			IF AW505PP = 1 THEN  !!! TA505PP = 1 Then
			!
			!C6 C7 C8 C9 C10 WD
			SetGO LaserProgReq, 153;
			MoveJ pA_505_1_N60_GM2,vProduction,fine,t3D_PFO\WObj:=wobj_A_GM2;
			rPFO_Welding;
			!
			!E6 WD
			SetGO PFOProgReq, 78;
			SetGO LaserProgReq, 140;
			MoveJ pA_505_3_N60_GM2,vProduction,fine,t3D_PFO\WObj:=wobj_A_GM2;
			rPFO_Welding;
			!
			ENDIF

			MoveJ pA_520_1_N60_GM2,vProduction,fine,t3D_PFO\WObj:=wobj_A_GM2;
			IF BW740PP = 1 THEN  !!!  TA520PP = 1 Then
			!
			!J3 WD
			SetGO PFOProgReq, 103;
			SetGO LaserProgReq, 140;
			MoveJ pA_520_1_N60_GM2,vProduction,fine,t3D_PFO\WObj:=wobj_A_GM2;
			rPFO_Welding;
			!
			!J8 WD
			SetGO PFOProgReq, 108;
			SetGO LaserProgReq, 140;
			MoveJ pA_520_4_N60_GM2,vProduction,fine,t3D_PFO\WObj:=wobj_A_GM2;
			rPFO_Welding;
			!
			ENDIF

			MoveJ pA_500_1_N60_GM2,vProduction,fine,t3D_PFO\WObj:=wobj_A_GM2;
			IF AW500PP = 1 THEN !!! TA500PP = 1 Then
			!
			!H6
			SetGO PFOProgReq, 100;
			SetGO LaserProgReq, 140;
			MoveJ pA_500_1_N60_GM2,vProduction,fine,t3D_PFO\WObj:=wobj_A_GM2;
			rPFO_Welding;
			!
			!F6 F7 F8 F9 F10
			SetGO LaserProgReq, 154;
			MoveJ pA_500_3_N60_GM2,vProduction,fine,t3D_PFO\WObj:=wobj_A_GM2;
			rPFO_Welding;
			!
			ENDIF

			MoveJ pA_Safe_1_N180_GM2, vProduction, z50, t3D_PFO\WObj:=wobj_A_GM2;

			!**************************************************
			!Trunnion at -180 degree
			!**************************************************
			MoveJ pA_500_1_N180_GM2,vProduction,fine,t3D_PFO\WObj:=wobj_A_GM2;
			IF AW500PP = 1 THEN !!! TA500PP = 1 Then
			!
			!N1 WD M3 M4 SP
			SetGO LaserProgReq, 155;
			MoveJ pA_500_1_N180_GM2,vProduction,fine,t3D_PFO\WObj:=wobj_A_GM2;
			rPFO_Welding;

			ENDIF

			! TA550
			MoveJ pA_550_1_N180_GM2,vProduction,fine,t3D_PFO\WObj:=wobj_A_GM2;
			IF AW550PP = 1 THEN  !!! TA550PP = 1 Then
			!
			!H2 H3 WD
			SetGO LaserProgReq, 166;
			MoveJ pA_550_1_N180_GM2,vProduction,fine,t3D_PFO\WObj:=wobj_A_GM2;
			rPFO_Welding;
			!
			!H1 WD
			SetGO PFOProgReq, 93;
			SetGO LaserProgReq, 140;
			MoveJ pA_550_2_N180_GM2,vProduction,fine,t3D_PFO\WObj:=wobj_A_GM2;
			rPFO_Welding;
			!
			!B13 B14 WD
			SetGO LaserProgReq, 167;
			MoveJ pA_550_3_N180_GM2,vProduction,fine,t3D_PFO\WObj:=wobj_A_GM2;
			rPFO_Welding;
			!
			!B15 B16 WD
			SetGO LaserProgReq, 168;
			MoveJ pA_550_4_N180_GM2,vProduction,fine,t3D_PFO\WObj:=wobj_A_GM2;
			rPFO_Welding;
			!
			!E1 WD
			SetGO PFOProgReq, 71;
			SetGO LaserProgReq, 140;
			MoveJ pA_550_5_N180_GM2,vProduction,fine,t3D_PFO\WObj:=wobj_A_GM2;
			rPFO_Welding;
			!
			!E2 E3 WD
			SetGO LaserProgReq, 169;
			MoveJ pA_550_6_N180_GM2,vProduction,fine,t3D_PFO\WObj:=wobj_A_GM2;
			rPFO_Welding;
			!
			!C5 WD
			SetGO PFOProgReq, 61;
			SetGO LaserProgReq, 140;
			MoveJ pA_550_7_N180_GM2,vProduction,fine,t3D_PFO\WObj:=wobj_A_GM2;
			rPFO_Welding;

			SetGO PFOProgReq, 22;
			SetGO LaserProgReq, 140;
			MoveJ pA_550_8_N180_GM2,vProduction,fine,t3D_PFO\WObj:=wobj_A_GM2;
			rPFO_Welding;
			!
			WaitTime 0.1;
			!
			SetGO PFOProgReq, 19;
			SetGO LaserProgReq, 140;
			MoveJ pA_550_8_N180_GM2,vProduction,fine,t3D_PFO\WObj:=wobj_A_GM2;
			rPFO_Welding;

			!A14 WD
			SetGO PFOProgReq, 14;
			SetGO LaserProgReq, 140;
			MoveJ pA_550_10_N180_GM2,vProduction,fine,t3D_PFO\WObj:=wobj_A_GM2;
			rPFO_Welding;
			!
			!A13
			SetGO PFOProgReq, 13;
			SetGO LaserProgReq, 140;
			MoveJ pA_550_12_N180_GM2,vProduction,fine,t3D_PFO\WObj:=wobj_A_GM2;
			rPFO_Welding;
			!
			!A4 WD
			SetGO PFOProgReq, 4;
			SetGO LaserProgReq, 140;
			MoveJ pA_550_13_N180_GM2,vProduction,fine,t3D_PFO\WObj:=wobj_A_GM2;
			rPFO_Welding;
			!
			!A1 WD
			SetGO PFOProgReq, 1;
			SetGO LaserProgReq, 140;
			MoveJ pA_550_14_N180_GM2,vProduction,fine,t3D_PFO\WObj:=wobj_A_GM2;
			rPFO_Welding;
			!
			!F5 WD
			SetGO PFOProgReq, 83;
			SetGO LaserProgReq, 140;
			MoveJ pA_550_15_N180_GM2,vProduction,fine,t3D_PFO\WObj:=wobj_A_GM2;
			rPFO_Welding;
			!
			ENDIF

			MoveJ pA_505_1_N180_GM2,vProduction,fine,t3D_PFO\WObj:=wobj_A_GM2;
			IF AW505PP = 1 THEN  !!! TA505PP = 1 Then
			!
			!L1 WD K3 K4 SP
			SetGO LaserProgReq, 160;
			MoveJ pA_505_1_N180_GM2,vProduction,fine,t3D_PFO\WObj:=wobj_A_GM2;
			rPFO_Welding;
			!
			ENDIF

			MoveJ pA_Safe_2_N180_GM2, vProduction, z200, t3D_PFO\WObj:=wobj_A_GM2;

			Reset PFOAirJet;
			Reset LaserRequest;
			AccSet 100,100;

			MoveAbsJ pA_Safe_N107\NoEOffs, vProduction, z200, t3D_PFO\WObj:=wobj0;
			MoveAbsJ pA_Safe_N069\NoEOffs, vProduction, z200, t3D_PFO\WObj:=wobj0;
			PulseDO\PLength:=2.0, WeldCompleted;
			MoveAbsJ pA_Safe_N031\NoEOffs, vProduction, z200, t3D_PFO\WObj:=wobj0;
			MoveAbsJ pA_Safe_P007\NoEOffs, vProduction, z200, t3D_PFO\WObj:=wobj0;
			MoveAbsJ pA_Unload\NoEOffs, vProduction, Fine, t3D_PFO\WObj:=wobj0;
			PulseDO\PLength:= 1.0, ToolAatLoadingPos;
		 IF ToolAChangeReq = 1 THEN
                 rTool_A_Change_Pos;
         ENDIF
			DeactUnit STN2;
			!WaitTime 0.25;
			!!
			!
			ClkStop clock_A_Weld_cycle;
			TPWrite "A Welding Cycle Time (ms) = " \Num:= ClkRead(clock_A_Weld_cycle)*1000;
			nA_Weld_Cycle_Time:= ClkRead(clock_A_Weld_cycle)*1000;
			SetGO TaskActive, 0;
	ENDPROC


ENDMODULE
